# EPICS substitutions: OLD/mc11/db/motor.substitutions
file "db/motor.db"
{

# ADDR ---> axis #
# NOTE ---> 2 asyn ports: 1) lowel comms ("P0"), and 2) Motor Record ("motor")
pattern
{ P,             M,                         MOTOR,   PORT,    ADDR, DESC,     DTYP,   MRES,     EGU,    PREC }
{ "XF:23ID2-BI", "{Diag:3-Ax:Y}Mtr", 	  "motor", "PO",    1,  "Diag:3 Y", asynMotor, "1.56e-3", "mm", 3 }
}
